TYPE ST_ClampingSafetyConfig :
STRUCT
    fMinimumAllowedPosition : LREAL;
    fModeSwitchVelocityMax : LREAL;

    // 绝对硬转矩上限预留；第一阶段关闭且不参与流程判断。
    bEnableHardMaxClampTorqueCheck : BOOL;
    fHardMaxClampTorquePercent : LREAL;
END_STRUCT
END_TYPE

(* stored: Version 1.1.0.1, ProductVersion 3.1.4026.20
   DUT ST_ClampingSafetyConfig: Id {c5f5f5bb-c6fd-45c9-83b1-234c8a4edfdf} *)
